// Implicitly generated code : DO NOT EDIT
FUNCTION CheckLRangeUnsigned : ULINT
VAR_INPUT
	value, lower, upper: ULINT;
END_VAR
VAR
    sMessageLow   : STRING := 'CheckLRangeUnsigned: Value too low (%d)';
    sMessageHigh  : STRING := 'CheckLRangeUnsigned: Value too high (%d)';
END_VAR

// Implicitly generated code : Only an Implementation suggestion
{noflow}
IF (value < lower) THEN
	CheckLRangeUnsigned := lower;
	// Log message
    ADSLOGLREAL(msgCtrlMask := ADSLOG_MSGTYPE_WARN,
               msgFmtStr   := sMessageLow,
               lrealArg     := TO_REAL(value));
ELSIF(value > upper) THEN
	CheckLRangeUnsigned := upper;
	// Log message
    ADSLOGLREAL(msgCtrlMask := ADSLOG_MSGTYPE_WARN,
               msgFmtStr   := sMessageHigh,
               lrealArg     := TO_REAL(value));
ELSE
	CheckLRangeUnsigned := value;
END_IF
{flow}

END_FUNCTION

(* stored: Version 1.1.0.1, ProductVersion 3.1.4024.11
   POU CheckLRangeUnsigned: Id {31ac514d-493f-43d8-8483-4f07aacc6999}, SpecialFunc CheckLRangeUnsigned *)
